PROGRAM MAIN
VAR
	n : UDINT := 5;
	result : ULINT;
	f : Factorial;
END_VAR

result := f(n);

END_PROGRAM

(* stored: Version 1.1.0.1, ProductVersion 3.1.4024.12
   POU MAIN: Id {3804045a-1986-48f3-bfb8-d7f2d97468a2}, SpecialFunc None *)
